			16#01: //16#2004-1
				MEMUtils.MemCpy(pbyDest:=ADR(DSO.NamurNe107) , pbySrc:=lcl_pointer+6 , dwSize:=1 );
				//MEMUtils.MemSet(pbyBuffer:=lcl_pointer+9 , byValue:=1 , dwSize:= 1);// Set Enable
				lcl_pointer[9]:=1;
			16#02: //16#2004-2
				MEMUtils.MemCpy(pbyDest:=ADR(DSO.Temperature)+2 , pbySrc:=lcl_pointer+4 , dwSize:=2 );
				MEMUtils.MemCpy(pbyDest:=ADR(DSO.Temperature) , pbySrc:=lcl_pointer+6 , dwSize:=2 );
				//MEMUtils.MemSet(pbyBuffer:=lcl_pointer+9 , byValue:=1 , dwSize:= 1);// Set Enable
				lcl_pointer[9]:=1;
			16#03: //16#2004-3
				MEMUtils.MemCpy(pbyDest:=ADR(DSO.Voltage)+2 , pbySrc:=lcl_pointer+4 , dwSize:=2 );
				MEMUtils.MemCpy(pbyDest:=ADR(DSO.Voltage) , pbySrc:=lcl_pointer+6 , dwSize:=2 );
				//MEMUtils.MemSet(pbyBuffer:=lcl_pointer+9 , byValue:=1 , dwSize:= 1);// Set Enable
				lcl_pointer[9]:=1;
			16#04: //16#2004-4
				MEMUtils.MemCpy(pbyDest:=ADR(DSO.Operational_Time_S)+2 , pbySrc:=lcl_pointer+4 , dwSize:=2 );
				MEMUtils.MemCpy(pbyDest:=ADR(DSO.Operational_Time_S) , pbySrc:=lcl_pointer+6 , dwSize:=2 );
				//MEMUtils.MemSet(pbyBuffer:=lcl_pointer+9 , byValue:=1 , dwSize:= 1);// Set Enable
				lcl_pointer[9]:=1;
			16#05: //16#2004-5
				MEMUtils.MemCpy(pbyDest:=ADR(DSO.Max_Temp)+2 , pbySrc:=lcl_pointer+4 , dwSize:=2 );
				MEMUtils.MemCpy(pbyDest:=ADR(DSO.Max_Temp) , pbySrc:=lcl_pointer+6 , dwSize:=2 );
				//MEMUtils.MemSet(pbyBuffer:=lcl_pointer+9 , byValue:=1 , dwSize:= 1);// Set Enable
				lcl_pointer[9]:=1;
			16#06: //16#2004-6
				MEMUtils.MemCpy(pbyDest:=ADR(DSO.Min_Temp)+2 , pbySrc:=lcl_pointer+4 , dwSize:=2 );
				MEMUtils.MemCpy(pbyDest:=ADR(DSO.Min_Temp) , pbySrc:=lcl_pointer+6 , dwSize:=2 );
				//MEMUtils.MemSet(pbyBuffer:=lcl_pointer+9 , byValue:=1 , dwSize:= 1);// Set Enable
				lcl_pointer[9]:=1;
			16#07: //16#2004-7
				MEMUtils.MemCpy(pbyDest:=ADR(DSO.Max_Voltage)+2 , pbySrc:=lcl_pointer+4 , dwSize:=2 );
				MEMUtils.MemCpy(pbyDest:=ADR(DSO.Max_Voltage) , pbySrc:=lcl_pointer+6 , dwSize:=2 );
				//MEMUtils.MemSet(pbyBuffer:=lcl_pointer+9 , byValue:=1 , dwSize:= 1);// Set Enable
				lcl_pointer[9]:=1;
			16#08: //16#2004-8
				MEMUtils.MemCpy(pbyDest:=ADR(DSO.Min_Voltage)+2 , pbySrc:=lcl_pointer+4 , dwSize:=2 );
				MEMUtils.MemCpy(pbyDest:=ADR(DSO.Min_Voltage) , pbySrc:=lcl_pointer+6 , dwSize:=2 );
				//MEMUtils.MemSet(pbyBuffer:=lcl_pointer+9 , byValue:=1 , dwSize:= 1);// Set Enable
				lcl_pointer[9]:=1;
		END_CASE;	
	END_IF;
	lcl_pointer:=lcl_pointer+Block_Size;
END_FOR;

END_FUNCTION_BLOCK

// 20 Program Organization Units/Level_0_Remote_IO/IFM/AL1340_UDFB
FUNCTION_BLOCK AL1340_UDFB
VAR
	i:INT;
	msgCounter:BYTE;
END_VAR

VAR_INPUT
	Acyclic_Response:cIFM_AL1342_Acyclic_Response;
	GW_TCP_State:ModbusTCPComState;
	
END_VAR


VAR_OUTPUT
	Port_Response:ARRAY[1..4] OF cIFM_AL1342_Acyclic_Response;
	Acyclic_Request:cIFM_AL1342_Acyclic_Request;
	Acyclic_Request_Active:BOOL;
	strTCPstate:STRING[30];
END_VAR
VAR_IN_OUT
	Port_Request:ARRAY[1..4] OF cIFM_AL1342_Acyclic_Request;
END_VAR

IF Acyclic_Response.Port>0 THEN
	Port_Response[Acyclic_Response.Port]:=Acyclic_Response;
	Port_Response[Acyclic_Response.Port].Port:=0;
	
END_IF;

IF Port_Request[i+1].Port =16#FF THEN
	msgCounter:=msgCounter+1;
	Port_Request[i+1].Port:=TO_WORD(i+1);
	Port_Request[i+1].User_ID:=msgCounter;
	Acyclic_Request:=Port_Request[i+1];
	Acyclic_Request_Active:=TRUE;
	
ELSE
	i:=(i+1) MOD 8;	
	Acyclic_Request_Active:=FALSE;
END_IF;



CASE GW_TCP_State OF
	ModbusTCPComState.OFF: strTCPstate:='OFF';
	ModbusTCPComState.CONNECTING: strTCPstate:='CONNECTING';
	ModbusTCPComState.CONNECTED: strTCPstate:='CONNECTED';
	ModbusTCPComState.DISCONNECTING: strTCPstate:='DISCONNECTING';
	ModbusTCPComState.SOCKET_ERROR: strTCPstate:='SOCKET_ERROR';
END_CASE

END_FUNCTION_BLOCK

// 20 Program Organization Units/Level_0_Remote_IO/IFM/AL1342_UDFB
FUNCTION_BLOCK AL1342_UDFB
VAR
	i:INT;
	msgCounter:BYTE;
END_VAR

VAR_INPUT
	Response:cIFM_AL1342_Acyclic_Response;
	
END_VAR


VAR_OUTPUT
	Port_Response:ARRAY[1..8] OF cIFM_AL1342_Acyclic_Response;
	Request:cIFM_AL1342_Acyclic_Request;
	Acyclic_Request:BOOL;
END_VAR
VAR_IN_OUT
	Port_Request:ARRAY[1..8] OF cIFM_AL1342_Acyclic_Request;
END_VAR

IF Response.Port>0 THEN
	Port_Response[Response.Port]:=Response;
	Port_Response[Response.Port].Port:=0;
	
END_IF;

IF Port_Request[i+1].Port =16#FF THEN
	msgCounter:=msgCounter+1;
	Port_Request[i+1].Port:=TO_WORD(i+1);
	Port_Request[i+1].User_ID:=msgCounter;
	Request:=Port_Request[i+1];
	Acyclic_Request:=TRUE;
	
ELSE
	i:=(i+1) MOD 8;	
	Acyclic_Request:=FALSE;
END_IF;

END_FUNCTION_BLOCK

// 20 Program Organization Units/Level_0_Remote_IO/Stride/MB0_RTD
FUNCTION_BLOCK MB0_RTD
VAR_INPUT
	GW_TCP_State:ModbusTCPComState;
	Device: REFERENCE TO cMB0_RTD;
	
	CH1: REFERENCE TO 	cSensor;
	CH1_Probe_Type:eMB0_RTD_Input_Type;
	CH2: REFERENCE TO 	cSensor;
	CH2_Probe_Type:eMB0_RTD_Input_Type;
	CH3: REFERENCE TO 	cSensor;
	CH3_Probe_Type:eMB0_RTD_Input_Type;
	CH4: REFERENCE TO 	cSensor;
	CH4_Probe_Type:eMB0_RTD_Input_Type;
	System_Units:eUnits;
END_VAR
VAR_OUTPUT
END_VAR
VAR
	Alarm:ARRAY[0..3] OF Analog_Alarm_UDFB;
END_VAR

CASE GW_TCP_State OF
	ModbusTCPComState.OFF: Device.strTCPstate:='OFF';
	ModbusTCPComState.CONNECTING: Device.strTCPstate:='CONNECTING';
	ModbusTCPComState.CONNECTED: Device.strTCPstate:='CONNECTED';
	ModbusTCPComState.DISCONNECTING: Device.strTCPstate:='DISCONNECTING';
	ModbusTCPComState.SOCKET_ERROR: Device.strTCPstate:='SOCKET_ERROR';
END_CASE





CASE System_Units OF
	eUnits.C:
		Device.TX.Holding_1218[0]:=eMB0_RTD_Units.C;
		Device.TX.Holding_1218[1]:=eMB0_RTD_Units.C;
		Device.TX.Holding_1218[2]:=eMB0_RTD_Units.C;
		Device.TX.Holding_1218[3]:=eMB0_RTD_Units.C;
	eUnits.F:
		Device.TX.Holding_1218[0]:=eMB0_RTD_Units.F;
		Device.TX.Holding_1218[1]:=eMB0_RTD_Units.F;
		Device.TX.Holding_1218[2]:=eMB0_RTD_Units.F;
		Device.TX.Holding_1218[3]:=eMB0_RTD_Units.F;
	eUnits.K:
		Device.TX.Holding_1218[0]:=eMB0_RTD_Units.k;
		Device.TX.Holding_1218[1]:=eMB0_RTD_Units.k;
		Device.TX.Holding_1218[2]:=eMB0_RTD_Units.k;
		Device.TX.Holding_1218[3]:=eMB0_RTD_Units.k;
END_CASE

Device.TX.Holding_31[0]:=CH1_Probe_Type;
Device.TX.Holding_31[1]:=CH1_Probe_Type;
Device.TX.Holding_31[2]:=CH1_Probe_Type;
Device.TX.Holding_31[3]:=CH1_Probe_Type;


CH1.EU:=TO_REAL(Device.RX.Holding_41[0])/10;
CH2.EU:=TO_REAL(Device.RX.Holding_41[1])/10;
CH3.EU:=TO_REAL(Device.RX.Holding_41[2])/10;
CH4.EU:=TO_REAL(Device.RX.Holding_41[3])/10;
IF NOT(Device.RX.Holding_50.0) THEN
	Alarm[0](
		Config:=CH1.Alarm_Config,
		EU:=CH1.EU,
		Debounce_Active:=CH1.Alarm_Config.Silence, 
		Status =>CH1.Status.eStatus,
		Percent_Alarm=>CH1.Alarm_Config.PCT_Alarm
		);
ELSE
	CH1.Status.eStatus:=eSensor_Status.Fault;
END_IF;
IF NOT(Device.RX.Holding_50.1) THEN
	Alarm[1](
		Config:=CH2.Alarm_Config,
		EU:=CH2.EU,
		Debounce_Active:=CH2.Alarm_Config.Silence, 
		Status =>CH2.Status.eStatus,
		Percent_Alarm=>CH2.Alarm_Config.PCT_Alarm
		);
ELSE
	CH2.Status.eStatus:=eSensor_Status.Fault;
END_IF;		
IF NOT(Device.RX.Holding_50.2) THEN
	Alarm[2](
		Config:=CH3.Alarm_Config,
		EU:=CH3.EU,
		Debounce_Active:=CH3.Alarm_Config.Silence, 
		Status =>CH3.Status.eStatus,
		Percent_Alarm=>CH3.Alarm_Config.PCT_Alarm
		);
ELSE
	CH3.Status.eStatus:=eSensor_Status.Fault;
END_IF;
IF NOT(Device.RX.Holding_50.3) THEN
	Alarm[3](
		Config:=CH4.Alarm_Config,
		EU:=CH4.EU,
		Debounce_Active:=CH4.Alarm_Config.Silence, 
		Status =>CH4.Status.eStatus,
		Percent_Alarm=>CH4.Alarm_Config.PCT_Alarm
		);
ELSE
	CH4.Status.eStatus:=eSensor_Status.Fault;
END_IF;	


IF NOT(GW_TCP_State=ModbusTCPComState.CONNECTED  OR GW_TCP_State=ModbusTCPComState.OFF) THEN
	CH1.Status.eStatus:=eSensor_Status.Offline;
	CH2.Status.eStatus:=eSensor_Status.Offline;
	CH3.Status.eStatus:=eSensor_Status.Offline;
	CH4.Status.eStatus:=eSensor_Status.Offline;
END_IF

END_FUNCTION_BLOCK

// 20 Program Organization Units/Level_0_Remote_IO/Stride/SIO_MB12CDR
FUNCTION_BLOCK SIO_MB12CDR
VAR_INPUT
	GW_TCP_State:ModbusTCPComState;
	Device : REFERENCE TO cSIO_MB12CDR;
	FIT_0:REFERENCE TO cBase_FIT;
	FIT_1:REFERENCE TO cBase_FIT;
	FIT_2:REFERENCE TO cBase_FIT;
	FIT_3:REFERENCE TO cBase_FIT;
END_VAR
VAR_OUTPUT
END_VAR
VAR
END_VAR

CASE GW_TCP_State OF
	ModbusTCPComState.OFF: Device.strTCPstate:='OFF';
	ModbusTCPComState.CONNECTING: Device.strTCPstate:='CONNECTING';
	ModbusTCPComState.CONNECTED: Device.strTCPstate:='CONNECTED';
	ModbusTCPComState.DISCONNECTING: Device.strTCPstate:='DISCONNECTING';
	ModbusTCPComState.SOCKET_ERROR: Device.strTCPstate:='SOCKET_ERROR';
END_CASE




Device.TX.Dout_31.0:=Device.Dout[0];
Device.TX.Dout_31.1:=Device.Dout[1];
Device.TX.Dout_31.2:=Device.Dout[2];
Device.TX.Dout_31.3:=Device.Dout[3];


Device.Din[0]:=Device.RX.Din_32.0;

END_FUNCTION_BLOCK

// 20 Program Organization Units/Level_0_Remote_IO/Wago/Wago_750_1405
FUNCTION Wago_750_1405 : bool
VAR_INPUT
	RX:WORD;
END_VAR
VAR_OUTPUT
	DI_1:BOOL;
	DI_2:BOOL;
	DI_3:BOOL;
	DI_4:BOOL;
	DI_5:BOOL;
	DI_6:BOOL;
	DI_7:BOOL;
	DI_8:BOOL;
	DI_9:BOOL;
	DI_10:BOOL;
	DI_11:BOOL;
	DI_12:BOOL;
	DI_13:BOOL;
	DI_14:BOOL;
	DI_15:BOOL;
	DI_16:BOOL;
END_VAR
VAR
END_VAR

DI_1:=RX.0;
DI_2:=RX.1;
DI_3:=RX.2;
DI_4:=RX.3;
DI_5:=RX.4;
DI_6:=RX.5;
DI_7:=RX.6;
DI_8:=RX.7;
DI_9:=RX.8;
DI_10:=RX.9;
DI_11:=RX.10;
DI_12:=RX.11;
DI_13:=RX.12;
DI_14:=RX.13;
DI_15:=RX.14;
DI_16:=RX.15;

END_FUNCTION

// 20 Program Organization Units/Level_0_Remote_IO/Wago/Wago_750_1504
FUNCTION Wago_750_1504 :Word;
VAR_INPUT
	DO_1:BOOL;
	DO_2:BOOL;
	DO_3:BOOL;
	DO_4:BOOL;
	DO_5:BOOL;
	DO_6:BOOL;
	DO_7:BOOL;
	DO_8:BOOL;
	DO_9:BOOL;
	DO_10:BOOL;
	DO_11:BOOL;
	DO_12:BOOL;
	DO_13:BOOL;
	DO_14:BOOL;
	DO_15:BOOL;
	DO_16:BOOL;
END_VAR
VAR
END_VAR

Wago_750_1504.0:=DO_1;
Wago_750_1504.1:=DO_2;
Wago_750_1504.2:=DO_3;
Wago_750_1504.3:=DO_4;
Wago_750_1504.4:=DO_5;
Wago_750_1504.5:=DO_6;
Wago_750_1504.6:=DO_7;
Wago_750_1504.7:=DO_8;
Wago_750_1504.8:=DO_9;
Wago_750_1504.9:=DO_10;
Wago_750_1504.10:=DO_11;
Wago_750_1504.11:=DO_12;
Wago_750_1504.12:=DO_13;
Wago_750_1504.13:=DO_14;
Wago_750_1504.14:=DO_15;
Wago_750_1504.15:=DO_16;

END_FUNCTION

// 20 Program Organization Units/Level_0_Remote_IO/Wago/Wago_750_496
FUNCTION Wago_750_496 : Bool
VAR_INPUT
	//Raw_Min:REAL:=(-765);
	//Raw_Max:REAL:=32763;
	RX:ARRAY[0..7] OF WORD;
END_VAR
VAR_OUTPUT
	AI_1:REAL;
	AI_1_PCT:REAL;
	AI_1_ma:REAL;
	AI_2:REAL;
	AI_2_PCT:REAL;
	AI_2_ma:REAL;
	AI_3:REAL;
	AI_3_PCT:REAL;
	AI_3_ma:REAL;
	AI_4:REAL;
	AI_4_PCT:REAL;
	AI_4_ma:REAL;
	AI_5:REAL;
	AI_5_PCT:REAL;
	AI_5_ma:REAL;
	AI_6:REAL;
	AI_6_PCT:REAL;
	AI_6_ma:REAL;
	AI_7:REAL;
	AI_7_PCT:REAL;
	AI_7_ma:REAL;
	AI_8:REAL;
	AI_8_PCT:REAL;
	AI_8_ma:REAL;
END_VAR
VAR
	PCT_Low:REAL:=-2.481;
	PCT_High:REAL:=106.26297;
	
	
	
END_VAR

AI_1:=TO_REAL(TO_INT(RX[0]));
AI_2:=TO_REAL(TO_INT(RX[1]));
AI_3:=TO_REAL(TO_INT(RX[2]));
AI_4:=TO_REAL(TO_INT(RX[3]));
AI_5:=TO_REAL(TO_INT(RX[4]));
AI_6:=TO_REAL(TO_INT(RX[5]));
AI_7:=TO_REAL(TO_INT(RX[6]));
AI_8:=TO_REAL(TO_INT(RX[7]));



AI_1_ma:=4.0+ (AI_1/1927);
AI_2_ma:=4.0+ (AI_2/1927);
AI_3_ma:=4.0+ (AI_3/1927);
AI_4_ma:=4.0+ (AI_4/1927);
AI_5_ma:=4.0+ (AI_5/1927);
AI_6_ma:=4.0+ (AI_6/1927);
AI_7_ma:=4.0+ (AI_7/1927);
AI_8_ma:=4.0+ (AI_8/1927);


AI_1_PCT:=Burkert_OSCAT_BASIC.SCALE_R(X:=AI_1_ma, I_LO:=3.60301, I_HI:=21.002 , O_LO:= PCT_Low, O_HI:=PCT_High );
AI_2_PCT:=Burkert_OSCAT_BASIC.SCALE_R(X:=AI_2_ma, I_LO:=3.60301, I_HI:=21.002 , O_LO:= PCT_Low, O_HI:=PCT_High );
AI_3_PCT:=Burkert_OSCAT_BASIC.SCALE_R(X:=AI_3_ma, I_LO:=3.60301, I_HI:=21.002 , O_LO:= PCT_Low, O_HI:=PCT_High );
AI_4_PCT:=Burkert_OSCAT_BASIC.SCALE_R(X:=AI_4_ma, I_LO:=3.60301, I_HI:=21.002 , O_LO:= PCT_Low, O_HI:=PCT_High );
AI_5_PCT:=Burkert_OSCAT_BASIC.SCALE_R(X:=AI_5_ma, I_LO:=3.60301, I_HI:=21.002 , O_LO:= PCT_Low, O_HI:=PCT_High );
AI_6_PCT:=Burkert_OSCAT_BASIC.SCALE_R(X:=AI_6_ma, I_LO:=3.60301, I_HI:=21.002 , O_LO:= PCT_Low, O_HI:=PCT_High );
AI_7_PCT:=Burkert_OSCAT_BASIC.SCALE_R(X:=AI_7_ma, I_LO:=3.60301, I_HI:=21.002 , O_LO:= PCT_Low, O_HI:=PCT_High );
AI_7_PCT:=Burkert_OSCAT_BASIC.SCALE_R(X:=AI_7_ma, I_LO:=3.60301, I_HI:=21.002 , O_LO:= PCT_Low, O_HI:=PCT_High );





// 16.000 ma = 30832 counts = 1927 counts / ma
// -765 loweset value =  -0.3969901 from base
// 0 = 4ma, -765 = -3.60301
//pct 0-100 iss 308.32 counts / percent, -765 counts = -2.4811, 32763 =102.26297

// max raw =- 32763 - 30832 = 1931 over
// max pct = 21.002ma

END_FUNCTION

// 20 Program Organization Units/Level_0_Remote_IO/Wago/Wago_750_555
FUNCTION Wago_750_555 : Array[0..3] of word
VAR_INPUT
	AO_1:REAL;
	AO_2:REAL;
	AO_3:REAL;
	AO_4:REAL;
END_VAR
VAR
END_VAR

Wago_750_555[0]:=TO_WORD(32767*(AO_1/100));
Wago_750_555[1]:=TO_WORD(32767*(AO_2/100));
Wago_750_555[2]:=TO_WORD(32767*(AO_3/100));
Wago_750_555[3]:=TO_WORD(32767*(AO_4/100));

END_FUNCTION

// 20 Program Organization Units/Level_1_Devices/Asi/ACV_ASI_CTRL_UDFB
FUNCTION_BLOCK ACV_ASI_CTRL_UDFB
VAR_INPUT
	FB:INT;
	CutOff:REAL:=0;
	LOCKOUT:BOOL:=FALSE;
	Online:BOOL:=TRUE;
	Error_PCT:REAL:=10;
	Error_Delay_S:INT:=10;
	LAS:BOOL:=TRUE;
	LDS:BOOL:=TRUE;
	LPS:BOOL:=TRUE;
	LPF:BOOL:=FALSE;
END_VAR
VAR_OUTPUT
	Status	:INT;
	Output	:INT;
END_VAR
VAR_IN_OUT
	//Valve	:ACV_DUT;
END_VAR
VAR
	//Output_TMP: REAL;
	//Scaled_Out: REAL;
	TON_1: TON;
	TOF_0: TOF;
	tmp_Output: REAL;
	FB_Real: REAL;
	Burkert_mode: Ton;
END_VAR

VAR_IN_OUT
	Valve:ASi_8694;
END_VAR

(* body of a kind this reader does not render *)

END_FUNCTION_BLOCK

// 20 Program Organization Units/Level_1_Devices/Asi/B8681_ASI_UDFB
FUNCTION_BLOCK B8681_ASI_UDFB
VAR_INPUT
	RX:BYTE;
	LAS:BOOL:=TRUE;
	LDS:BOOL:=TRUE;
	LPS:BOOL:=TRUE;
	LPF:BOOL:=FALSE;
END_VAR
VAR_OUTPUT
	TX:BYTE;
END_VAR
VAR
	lcl_status: BYTE;
END_VAR
VAR_IN_OUT
	Valve:B8691_Asi_DUT;
END_VAR
VAR // added by the converter: edge detectors and wires of the graphical bodies
    _w1, _w2, _w3 : ANY;
END_VAR

_w1 := (Valve.Mode=e_8681_Modes.Auto) AND (Valve.PLC_CMD=e_8681_Modes.Upper_Drain) OR (Valve.Mode=e_8681_Modes.Upper_Drain);
_w2 := SEL(_w1, SEL((Valve.Mode=e_8681_Modes.Auto) AND (Valve.PLC_CMD=e_8681_Modes.Lower_Drain) OR (Valve.Mode=e_8681_Modes.Lower_Drain), SEL((Valve.Mode=e_8681_Modes.Auto) AND (Valve.PLC_CMD=e_8681_Modes.Open) OR (Valve.Mode=e_8681_Modes.Open), 0, 1), 2), 4);
TX := _w2;
BURKERT_OSCAT_BASIC.WORD_OF_BYTE\(B1 := _w2, B0 := RX, WORD_OF_BYTE => _w3);
Valve.Status := _w3;
Valve.Status1 := SEL(LPF, SEL(LDS AND NOT LAS, SEL(NOT LAS, SEL(RX.2, SEL(_w1, SEL(RX.0, SEL(RX.1, eB8681_Status.Unknown, eB8681_Status.Open), eB8681_Status.Blocked), eB8681_Status.Upper_Drain), eB8681_Status.Lower_Drain), eB8681_Status.Missing), eB8681_Status.Detected), eB8681_Status.P_Fault);

END_FUNCTION_BLOCK

// 20 Program Organization Units/Level_1_Devices/Asi/BCV_ASI_CTRL_UDFB
FUNCTION_BLOCK BCV_ASI_CTRL_UDFB
VAR_INPUT
	OL:BOOL;
	CL:BOOL;
	LOCKOUT:BOOL:=FALSE;
	Online:BOOL:=TRUE;
	LAS:BOOL:=TRUE;
	LDS:BOOL:=TRUE;
	LPS:BOOL:=TRUE;
	LPF:BOOL:=FALSE;

END_VAR
VAR_OUTPUT
	Output	:BOOL;
END_VAR
VAR_IN_OUT
	BCV:cBCV;
END_VAR
VAR
	
	Test: BOOL;
	GEN_PULSE_0: Burkert_OSCAT_BASIC.GEN_PULSE;
	Burkert_Open_Ton: TON;
END_VAR

(* body of a kind this reader does not render *)

END_FUNCTION_BLOCK

// 20 Program Organization Units/Level_1_Devices/Base_Functions/Basic_ACV_UDFB
FUNCTION_BLOCK Basic_ACV_UDFB
VAR_INPUT
	FB:REAL;
	CutOff:REAL;
	LockOut_NC:BOOL;
	Online:BOOL;
	Error_PCT:REAL;
	Error_Delay_S:INT;
	Permissive_NC:BOOL;
	Position_Hold:BOOL:=FALSE;
END_VAR
VAR_OUTPUT
	Status	:INT;
	Output	:REAL;
	Active:BOOL;
	oldPos:REAL;
END_VAR
VAR_IN_OUT
	Valve	:cACV;
END_VAR
VAR
	TON_1: TON;
	TOF_0: TOF;
	DataOk:BOOL:=FALSE;
	tIndex:INT:=0;
	PosArray:ARRAY[0..4] OF REAL;
	lcl_Status:eACV_Status;
	Control_Error:REAL;
	PosChange:REAL;
	Active_TOf:TOF;
	Trend:ARRAY[0..14] OF REAL;
	//Trend_Detect:Burkert_Oscat_Basic.TREND;
	
	TOF_1: TOF;
	Active_TON:Ton;
END_VAR

(* body of a kind this reader does not render *)

END_FUNCTION_BLOCK

// 20 Program Organization Units/Level_1_Devices/Base_Functions/Basic_BCV_UDFB
FUNCTION_BLOCK Basic_BCV_UDFB
VAR_INPUT
	OL:BOOL;
	CL:BOOL;
	LOCKOUT:BOOL;
	Online:BOOL;
	Interlock:BOOL;
END_VAR

VAR_OUTPUT
	Output	:BOOL;
	Output_2	:BOOL;
END_VAR

VAR_IN_OUT
	BCV	:cBCV;
END_VAR

VAR
	Pulse:Burkert_Oscat_basic.GEN_SQ;
	TON_0:Ton;
	TOF_0:TOF;
END_VAR


	

Output:=Eval_Output();
Output_2:=NOT(Output);

IF BCV.Mode.eMode=eBCV_Modes.Simulate THEN
	BCV.Ready:=TRUE;
	IF Output THEN 
		BCV.Status.eStatus:=eBCV_Status.A_Open;	
	ELSE
		BCV.Status.eStatus:=eBCV_Status.A_Closed;
	END_IF
ELSE	
	BCV.Ready:=Eval_Ready();
	BCV.Status.eStatus:= Eval_Status();
END_IF;

END_FUNCTION_BLOCK

// 20 Program Organization Units/Level_1_Devices/Base_Functions/Basic_FIT
FUNCTION_BLOCK Basic_FIT
VAR_INPUT
	//Count:DWORD;
	//Frequency:REAL;
	//Raw_Count_16Bit:BOOL;
	Rate_Units:eUnits;
	Volume_Units:eUnits;
	
	FIT:REFERENCE TO cBase_FIT;
END_VAR

VAR_OUTPUT
	Reset:BOOL;
END_VAR

VAR
	Analog_Alarm:Analog_Alarm_UDFB;
	R_Trig_0: R_Trig;
	COUNT_REAL: LREAL;
	Total:LREAL;
	FREQUENCY_REAL: REAL;
	Rate_Sec:REAL;
	High_Word:Word;
	ALARM_1_0: BURKERT_OSCAT_BASIC.ALARM_2;
	hihi: BOOL;
	hi: BOOL;
	lolo: BOOL;
	LO: BOOL;
	Alarm_Debounce: TON;
	TON_0: TON;
END_VAR
VAR_IN_OUT
	
END_VAR

(* body of a kind this reader does not render *)

END_FUNCTION_BLOCK

// 20 Program Organization Units/Level_1_Devices/Base_Functions/BCV_CTRL_UDFB
FUNCTION_BLOCK BCV_CTRL_UDFB
VAR_INPUT
	OL:BOOL;
	CL:BOOL;
	LOCKOUT:BOOL:=FALSE;
	Online:BOOL:=TRUE;
	Interlock:BOOL;
END_VAR

VAR_OUTPUT
	Output	:BOOL;
	Output_2	:BOOL;
END_VAR

VAR_IN_OUT
	BCV	:cBCV;
END_VAR

VAR  
	Pulse_0: Burkert_OSCAT_BASIC.GEN_SQ;
	
END_VAR

(* body of a kind this reader does not render *)

END_FUNCTION_BLOCK

// 20 Program Organization Units/Level_1_Devices/Base_Functions/Contactor_Control_UDFB
FUNCTION_BLOCK Contactor_Control_UDFB
VAR_INPUT
	Allow_Reverse:BOOL;
	Inhibit_FWD:BOOL:=FALSE;
	Inhibit_Rev:BOOL:=FALSE;
	Bump_Duration:TIME:=T#1S;
END_VAR
VAR_OUTPUT
	Q_FWD:BOOL;
	Q_REV:Bool;
END_VAR
VAR
	//F_TRIG_0: F_trig;
	TP_0: TP;
	F_TRIG_1: F_trig;
	TP_1: TP;
END_VAR
VAR_IN_OUT
	Contactor:Contactor_DUT;
END_VAR
VAR // added by the converter: edge detectors and wires of the graphical bodies
    _w1, _w2, _w4, _w5, _w6, _w7, _w8, _w10, _w11, _w12 : BOOL;
    _w3, _w9 : ANY;
END_VAR

_w1 := Contactor.Mode.eMode = Contactor_Modes.Auto;
_w2 := _w1 AND Contactor.PLC_CMD_FWD;
_w3 := SEL(_w2, Contactor_Status.OFF, Contactor_Status.Auto_FWD);
_w4 := Contactor.Mode.eMode = Contactor_Modes.Fwd;
TP_1(IN := Contactor.Mode.eMode = Contactor_Modes.Bump_FWD, PT := Bump_Duration); // TP
_w5 := _w4 OR TP_1.Q;
_w6 := _w2 OR _w5;
_w7 := _w6 AND NOT Inhibit_FWD AND NOT (Contactor.Mode.eMode=Contactor_Modes.Disabled);
Contactor.Q1 := _w7;
Q_FWD := _w7;
_w8 := _w1 AND Contactor.PLC_CMD_Rev;
_w9 := SEL(_w8, SEL((_w2 OR _w5) AND Inhibit_FWD, SEL(_w5, _w3, Contactor_Status.Manual_FWD), Contactor_Status.FWD_Limit), Contactor_Status.Auto_Rev);
_w10 := Contactor.Mode.eMode = Contactor_Modes.Rev;
TP_0(IN := Contactor.Mode.eMode = Contactor_Modes.Bump_REV, PT := Bump_Duration); // TP
_w11 := _w10 OR TP_0.Q;
Contactor.Status := SEL((_w8 OR _w11) AND Inhibit_REV, SEL(_w11, _w9, Contactor_Status.Manual_Rev), Contactor_Status.REV_Limit);
_w12 := (NOT _w6 AND (_w8 OR _w11) AND Allow_Reverse) AND NOT Inhibit_REV AND NOT (Contactor.Mode.eMode=Contactor_Modes.Disabled);
Q_Rev := _w12;
Contactor.Q2 := _w12;
F_TRIG_1(CLK := TP_1.Q OR TP_0.Q); // F_trig

END_FUNCTION_BLOCK

// 20 Program Organization Units/Level_1_Devices/Base_Functions/DO_UDFB
FUNCTION_BLOCK DO_UDFB
VAR_INPUT
	Lockout_NC:BOOL;
	Permisive_NC:BOOL;
	OnLine:Bool;
	
	
END_VAR
VAR_OUTPUT
	Q:BOOL;
END_VAR
VAR
END_VAR
VAR_IN_OUT
	Dout:Do_DUT;
END_VAR
VAR // added by the converter: edge detectors and wires of the graphical bodies
    _w1, _w2, _w3 : BOOL;
END_VAR

_w1 := SEL(Dout.Mode.eMode=DO_modes.Forced_On, False, True);
_w2 := Permisive_NC AND ((Dout.Mode.eMode=DO_modes.Auto) AND Dout.PLC_CMD);
_w3 := Lockout_NC AND (_w2 OR SEL(Dout.Mode.eMode=DO_modes.Forced_Off, _w1, False));
Dout.Q := _w3;
Q := _w3;
dout.Status := SEL(NOT OnLine, SEL(LockOut_NC, Do_Status.LOCKED_OUT, SEL(_w2, SEL(Dout.Mode.eMode=DO_modes.Forced_Off, SEL(_w1, SEL(permisive_NC, Do_Status.Interlocked, Do_Status.OFF), Do_Status.Forced_On), Do_Status.Forced_OFF), Do_Status.On)), Do_Status.OFFLINE);
Dout.Ready := Online AND (Dout.Mode.eMode=Do_modes.Auto);

END_FUNCTION_BLOCK

// 20 Program Organization Units/Level_1_Devices/Base_Functions/LS_UDFB
FUNCTION_BLOCK LS_UDFB
VAR_INPUT
	Wired_NC:BOOL;
	On_Delay_ms:UINT;
	Off_Delay_ms:UINT;
	Alarm_Dry:BOOL;
	Alarm_Wet:BOOL;
	Raw:BOOL;
	Device: REFERENCE TO DI_DUT;
	Card_OK:BOOL:=TRUE;
	
END_VAR
VAR_OUTPUT
END_VAR
	

VAR
	TON_0:TON;
	TOF_0:TOF;
	LCL_raw:Bool;
END_VAR

VAR_IN_OUT
	//Device:DI_DUT;
END_VAR

Device.Raw:=Raw;
CASE Device.MODE.eMode OF 
	DI_Modes.Auto: 			LCL_Raw:=Device.Raw;
	DI_Modes.Forced_Off:	LCL_Raw:=FALSE;
	DI_Modes.Forced_On:		LCL_Raw:=TRUE;
END_CASE

TON_0(PT:=(TO_TIME(On_Delay_ms)),IN:=LCL_RAW);
TOF_0(PT:=(TO_TIME(Off_Delay_ms)),IN:=TON_0.Q,Q=>Device.Q);


IF Wired_NC THEN
	Device.Status.eStatus:=SEL(Device.Q,DI_Status.Liquid_Detected,DI_Status.No_Liquid_Detected);
ELSE
	Device.Status.eStatus:=SEL(Device.Q,DI_Status.NO_Liquid_Detected,DI_Status.Liquid_Detected);
END_IF;

IF Alarm_Dry AND Device.Status.eStatus=DI_Status.NO_Liquid_Detected THEN
	Device.Status.eStatus:=DI_Status.No_Liquid_Detected_Alarm;
END_IF;

IF Alarm_Wet AND Device.Status.eStatus=DI_Status.Liquid_Detected THEN
	Device.Status.eStatus:=DI_Status.Liquid_Detected_Alarm;
END_IF;
IF NOT(Card_Ok) AND Device.MODE.eMode=DI_Modes.Auto THEN Device.Status.eStatus:=DI_Status.IO_Fault; END_IF;

END_FUNCTION_BLOCK
